// TIA Portal V17 export
// export: Created 2022-07-28T18:02:47.2254951Z, ExportSetting None, DisplayName Totally Integrated Automation Portal, DisplayVersion V17, DisplayName TIA Portal Openness, DisplayVersion V17, DisplayName TIA Portal Teamcenter Gateway, DisplayVersion V17, DisplayName TIA Portal Version Control Interface, DisplayVersion V17, DisplayName TIA Portal Test Suite Advanced, DisplayVersion V17, DisplayName SINAMICS Startdrive Advanced, DisplayVersion V17, DisplayName SINAMICS DCC, DisplayVersion V17, DisplayName SINAMICS Startdrive G130, G150, S120, S150, SINAMICS MV, S210, DisplayVersion V17, DisplayName SINAMICS Startdrive G110M, G120, G120C, G120D, G120P, G115D, DisplayVersion V17, DisplayName STEP 7 Professional, DisplayVersion V17, DisplayName SIMATIC Energy Suite, DisplayVersion V17, DisplayName STEP 7 CFC, DisplayVersion V17, DisplayName STEP 7 Safety, DisplayVersion V17, DisplayName WinCC Advanced / Unified PC, DisplayVersion V17, DisplayName SIMATIC Visualization Architect, DisplayVersion V17
FUNCTION_BLOCK "Internal_H01_FB"   // FB8, SCL
TITLE = InternalH01
{ S7_Optimized_Access := 'TRUE' }
// Proccess signals from fuses, safety and others internal devices
// stored: MemoryReserve 100, SetENOAutomatically false
   VAR_INPUT
      I_CmdGeneralReset { ExternalAccessible := 'False'; ExternalVisible := 'False'; ExternalWritable := 'False'} : Bool;   // 0 ⮥ 1 = Input general reset ERROR/Interlocks
      IR_CycleTime { ExternalAccessible := 'False'; ExternalVisible := 'False'; ExternalWritable := 'False'} : Real := 0.0;   // Time of last PLC cycle, sec
      I_Initialization { ExternalAccessible := 'False'; ExternalVisible := 'False'; ExternalWritable := 'False'} : Bool := FALSE;   // 1 = Restart PLC is active (First scan)
      I_One_1s { ExternalAccessible := 'False'; ExternalVisible := 'False'; ExternalWritable := 'False'} : Bool;   // 1 = One cycle per one seccond pulse
      I_KV_Ok { ExternalAccessible := 'False'; ExternalVisible := 'False'; ExternalWritable := 'False'} : Bool;   // Напруга 400VAC в нормі -KV1
      I_QF_Trans_Ok { ExternalAccessible := 'False'; ExternalVisible := 'False'; ExternalWritable := 'False'} : Bool;   // Автомат захисту трансформатора -Q1
      I_QF_Oper230_Ok { ExternalAccessible := 'False'; ExternalVisible := 'False'; ExternalWritable := 'False'} : Bool;   // Розподільчий автомат оперативної напруги 230 V AC -F1
      I_QF_Oper24_Ok { ExternalAccessible := 'False'; ExternalVisible := 'False'; ExternalWritable := 'False'} : Bool;   // Живлення оперативної напруги 24 V DC -F2
      I_QF_Saf_Ok { ExternalAccessible := 'False'; ExternalVisible := 'False'; ExternalWritable := 'False'} : Bool;   // Живлення кіл безпеки -F3
      I_QF_KM_Ok { ExternalAccessible := 'False'; ExternalVisible := 'False'; ExternalWritable := 'False'} : Bool;   // Живлення котушок контакторів -F4
      I_QF_Gas_Ok { ExternalAccessible := 'False'; ExternalVisible := 'False'; ExternalWritable := 'False'} : Bool;   // Живлення сигналізатора загазованості -F5
      I_QF_VlvSaf_Ok { ExternalAccessible := 'False'; ExternalVisible := 'False'; ExternalWritable := 'False'} : Bool;   // Живлення відсічного клапана -F6
      I_QF_Spare_Ok { ExternalAccessible := 'False'; ExternalVisible := 'False'; ExternalWritable := 'False'} : Bool;   // Резерв -F7
   END_VAR
   VAR_OUTPUT
      QW_STW { ExternalWritable := 'False'} : Word;   // Status for HMI
      Q_Reset { ExternalAccessible := 'False'; ExternalVisible := 'False'; ExternalWritable := 'False'} : Bool;   // 1 = Reset external err
      Q_SomeErr { ExternalAccessible := 'False'; ExternalVisible := 'False'; ExternalWritable := 'False'} : Bool;   // 1 = Some err occured
      Q_KV_Ok { ExternalAccessible := 'False'; ExternalVisible := 'False'; ExternalWritable := 'False'} : Bool;   // Напруга 400VAC в нормі -KV1
      Q_QF_Trans_Ok { ExternalAccessible := 'False'; ExternalVisible := 'False'; ExternalWritable := 'False'} : Bool;   // Автомат захисту трансформатора -Q1
      Q_QF_Oper230_Ok { ExternalAccessible := 'False'; ExternalVisible := 'False'; ExternalWritable := 'False'} : Bool;   // Розподільчий автомат оперативної напруги 230 V AC -F1
      Q_QF_Oper24_Ok { ExternalAccessible := 'False'; ExternalVisible := 'False'; ExternalWritable := 'False'} : Bool;   // Живлення оперативної напруги 24 V DC -F2
      Q_QF_Saf_Ok { ExternalAccessible := 'False'; ExternalVisible := 'False'; ExternalWritable := 'False'} : Bool;   // Живлення кіл безпеки -F3
      Q_QF_KM_Ok { ExternalAccessible := 'False'; ExternalVisible := 'False'; ExternalWritable := 'False'} : Bool;   // Живлення котушок контакторів -F4
      Q_QF_Gas_Ok { ExternalAccessible := 'False'; ExternalVisible := 'False'; ExternalWritable := 'False'} : Bool;   // Живлення сигналізатора загазованості -F5
      Q_QF_VlvSaf_Ok { ExternalAccessible := 'False'; ExternalVisible := 'False'; ExternalWritable := 'False'} : Bool;   // Живлення відсічного клапана -F6
      Q_QF_Spare_Ok { ExternalAccessible := 'False'; ExternalVisible := 'False'; ExternalWritable := 'False'} : Bool;   // Резерв -F7
   END_VAR
   VAR_IN_OUT
      II_CMD : Int;   // Command from HMI for current box
   END_VAR
   VAR
      s_KV_Err { ExternalAccessible := 'False'; ExternalVisible := 'False'; ExternalWritable := 'False'} : Bool;   // Напруга 400VAC в нормі -KV1
      s_QF_Trans_Err { ExternalAccessible := 'False'; ExternalVisible := 'False'; ExternalWritable := 'False'} : Bool;   // Автомат захисту трансформатора -Q1
      s_QF_Oper230_Err { ExternalAccessible := 'False'; ExternalVisible := 'False'; ExternalWritable := 'False'} : Bool;   // Розподільчий автомат оперативної напруги 230 V AC -F1
      s_QF_Oper24_Err { ExternalAccessible := 'False'; ExternalVisible := 'False'; ExternalWritable := 'False'} : Bool;   // Живлення оперативної напруги 24 V DC -F2
      s_QF_Saf_Err { ExternalAccessible := 'False'; ExternalVisible := 'False'; ExternalWritable := 'False'} : Bool;   // Живлення кіл безпеки -F3
      s_QF_KM_Err { ExternalAccessible := 'False'; ExternalVisible := 'False'; ExternalWritable := 'False'} : Bool;   // Живлення котушок контакторів -F4
      s_QF_Gas_Err { ExternalAccessible := 'False'; ExternalVisible := 'False'; ExternalWritable := 'False'} : Bool;   // Живлення сигналізатора загазованості -F5
      s_QF_VlvSaf_Err { ExternalAccessible := 'False'; ExternalVisible := 'False'; ExternalWritable := 'False'} : Bool;   // Живлення відсічного клапана -F6
      s_QF_Spare_Err { ExternalAccessible := 'False'; ExternalVisible := 'False'; ExternalWritable := 'False'} : Bool;   // Резерв -F7
      s_TP_Reset { ExternalAccessible := 'False'; ExternalVisible := 'False'; ExternalWritable := 'False'} : "Lib_FB_Timer_TP_Simple";
   END_VAR
   VAR_TEMP
      t_ResetHMI : Bool;   // Reset from HMI
      t_ResetLogic : Bool;   // Reset for logic
      t_SomeErr : Bool;   // 1 = Some err occured
      ti_LogicCMD : Int;   // CMD for logic
      tw_STW : Word;   // Status for HMI
   END_VAR
BEGIN
   REGION Initialization
       IF #II_CMD <> 0
       THEN
           #ti_LogicCMD := #II_CMD;
           #II_CMD := 0;
       ELSE
           #ti_LogicCMD := 0;
       END_IF;

       #t_ResetHMI := false;
       #tw_STW := w#16#0;
   END_REGION

   REGION Reset for logic
       //Reset from HMI
       CASE #ti_LogicCMD OF
           31..32:  //Reset
               #t_ResetHMI := true;
           ELSE  // Statement section ELSE
               ;
       END_CASE;

       //Reset for logic
       #t_ResetLogic := #t_ResetHMI
       OR #I_CmdGeneralReset;

       #s_TP_Reset(IR_CycleTime:=#IR_CycleTime,
                   IB_StartTimerInput:=#t_ResetLogic,
                   IR_SpTime:=2.0,
                   QB_TimerOut=>#t_ResetLogic);

   END_REGION

   REGION Catch errors
       #s_KV_Err := (NOT #I_KV_Ok
       OR (#s_KV_Err
       AND NOT #t_ResetLogic)) 
       AND NOT #I_Initialization;

       #s_QF_Trans_Err := (NOT #I_QF_Trans_Ok
       OR (#s_QF_Trans_Err
       AND NOT #t_ResetLogic))
       AND NOT #I_Initialization;

       #s_QF_Oper230_Err := (NOT #I_QF_Oper230_Ok
       OR (#s_QF_Oper230_Err
       AND NOT #t_ResetLogic))
       AND NOT #I_Initialization;

       #s_QF_Oper24_Err := (NOT #I_QF_Oper24_Ok
       OR (#s_QF_Oper24_Err
       AND NOT #t_ResetLogic))
       AND NOT #I_Initialization;

       #s_QF_Saf_Err := (NOT #I_QF_Saf_Ok
       OR (#s_QF_Saf_Err
       AND NOT #t_ResetLogic))
       AND NOT #I_Initialization;

       #s_QF_KM_Err := (NOT #I_QF_KM_Ok
       OR (#s_QF_KM_Err
       AND NOT #t_ResetLogic))
       AND NOT #I_Initialization;

       #s_QF_Gas_Err := (NOT #I_QF_Gas_Ok
       OR (#s_QF_Gas_Err
       AND NOT #t_ResetLogic))
       AND NOT #I_Initialization;

       #s_QF_VlvSaf_Err := (NOT #I_QF_VlvSaf_Ok
       OR (#s_QF_VlvSaf_Err
       AND NOT #t_ResetLogic))
       AND NOT #I_Initialization;

       #s_QF_Spare_Err := (NOT #I_QF_Spare_Ok
       OR (#s_QF_Spare_Err
       AND NOT #t_ResetLogic))
       AND NOT #I_Initialization;
   END_REGION

   REGION Write STW
       //Some err occured
       #t_SomeErr := #s_KV_Err
       OR #s_QF_Trans_Err
       OR #s_QF_Oper230_Err
       OR #s_QF_Oper24_Err
       OR #s_QF_Saf_Err
       OR #s_QF_KM_Err
       OR #s_QF_Gas_Err
       OR #s_QF_VlvSaf_Err
       OR #s_QF_Spare_Err;

       //Write err to STW
       #tw_STW.%X0 := #t_SomeErr;
       #tw_STW.%X1 := #s_KV_Err;
       #tw_STW.%X2 := #s_QF_Trans_Err;
       #tw_STW.%X3 := #s_QF_Oper230_Err;
       #tw_STW.%X4 := #s_QF_Oper24_Err;
       #tw_STW.%X5 := #s_QF_Saf_Err;
       #tw_STW.%X6 := #s_QF_KM_Err;
       #tw_STW.%X7 := #s_QF_Gas_Err;
       #tw_STW.%X8 := #s_QF_VlvSaf_Err;
       #tw_STW.%X9 := #s_QF_Spare_Err;
   END_REGION

   REGION Write outs
       #QW_STW := #tw_STW;
       #Q_Reset := #t_ResetLogic;
       #Q_SomeErr := #t_SomeErr;
       #Q_KV_Ok := NOT #s_KV_Err;
       #Q_QF_Trans_Ok := NOT #s_QF_Trans_Err;
       #Q_QF_Oper230_Ok := NOT #s_QF_Oper230_Err;
       #Q_QF_Oper24_Ok := NOT #s_QF_Oper24_Err;
       #Q_QF_Saf_Ok := NOT #s_QF_Saf_Err;
       #Q_QF_KM_Ok := NOT #s_QF_KM_Err;
       #Q_QF_Gas_Ok := NOT #s_QF_Gas_Err;
       #Q_QF_VlvSaf_Ok := NOT #s_QF_VlvSaf_Err;
       #Q_QF_Spare_Ok := NOT #s_QF_Spare_Err;
   END_REGION
END_FUNCTION_BLOCK
